// TIA Portal V19 export
TYPE "C501_STU_IF_BBI_TYPIC"
   STRUCT
      WRE { ExternalAccessible := 'False'; ExternalVisible := 'False'; ExternalWritable := 'False'} : USInt;   // Actueel actief regime
   END_STRUCT;
END_TYPE
